FUNCTION F_RadToDeg : LREAL
VAR_INPUT
	fRad : LREAL;
END_VAR
VAR
END_VAR

F_RadToDeg := fRad * (180/PI);

END_FUNCTION

(* stored: Version 1.1.0.1, ProductVersion 3.1.4024.10
   POU F_RadToDeg: Id {b20df42b-409d-413f-bfa5-4422ba4a12e6}, SpecialFunc None *)
